FUNCTION "LAxisCtrlApcFr_UnpubAxisStatusDriveCommunicationOK" : Bool
TITLE = LAxisCtrl_UnpubAxisPosition
{ S7_Optimized_Access := 'TRUE' }
AUTHOR : 'tech.team.motioncontrol@siemens.com'
FAMILY : AxisCtrl
VERSION : 1.2
//Support: tech.team.motioncontrol@siemens.com
   VAR_INPUT
      axis : DB_ANY;   // Axis specification
   END_VAR

   VAR_TEMP
      tempRefSpeedAxis {InstructionName := 'TO_SpeedAxis'; LibVersion := '8.0'} : REF_TO TO_SpeedAxis;   // Temporary reference of the technology object type TO_SpeedAxis
   END_VAR


BEGIN
	// Read axis parameter
	#tempRefSpeedAxis ?= #axis;

	IF (#tempRefSpeedAxis <> NULL) THEN
	    // Axis type is TO_SpeedAxis or TO_PositioningAxis or TO_SynchronousAxis
	    #LAxisCtrlApcFr_UnpubAxisStatusDriveCommunicationOK := #tempRefSpeedAxis^.StatusDrive.CommunicationOK;
	ELSE
	    // Invalid TO specification
	    #LAxisCtrlApcFr_UnpubAxisStatusDriveCommunicationOK := FALSE;
	END_IF;

END_FUNCTION

